INTERFACE I_Devices

METHOD M_CyclicLogic : HRESULT
END_METHOD

END_INTERFACE

(* stored: Version 1.1.0.1
   Itf I_Devices: Id {5ce81993-9a4e-487b-93ae-e57eed0e1a2d}
   Method M_CyclicLogic: Id {457039af-a69b-4f5f-a08e-36c991da531e} *)
